TYPE ACRMemoryTimeEvents :
STRUCT
	_Values : ARRAY [0..GCL.cMemoryEventsMidMAX] OF ACRMemoryTimeEvent;
END_STRUCT
END_TYPE

(* stored: Version 1.1.0.1, ProductVersion 3.1.4020.12
   DUT ACRMemoryTimeEvents: Id {adad75c6-33ef-40fa-a0b6-eb6a980f407b} *)
